INTERFACE I_InputPorts

METHOD PUBLIC Accept
VAR_INPUT
	Visitor : I_InputPortVisitor;
END_VAR
END_METHOD

METHOD PUBLIC AddDataAsInputPort : I_InputPort
VAR_INPUT
	Name : T_MAXSTRING;
	Data : I_Datatype;
END_VAR
END_METHOD

METHOD AddInputPort
VAR_INPUT
	InputPort : I_InputPort;
END_VAR
END_METHOD

METHOD PUBLIC TryGetInputPortByName : BOOL
VAR_INPUT
	Name : T_MAXSTRING;
	Destination : REFERENCE TO I_InputPort;
END_VAR
END_METHOD

END_INTERFACE

(* stored: Version 1.1.0.1, ProductVersion 3.1.4024.12
   Itf I_InputPorts: Id {b540daf3-61f2-4ef3-ad34-4bde554d65b6}
   Method Accept: Id {5bb2f9c8-2ef3-400e-ab86-bca85c02c626}
   Method AddDataAsInputPort: Id {ae463917-1501-47bf-b38f-f3111fdbb0d8}
   Method AddInputPort: Id {135eb44b-cbc4-0e2f-0792-05757aacdb77}
   Method TryGetInputPortByName: Id {a21ad5ef-ba3e-0598-3880-d9f06b97f2a5} *)
